(* PLC project actuator, TNI-Software ControlBuild 4.00.17 *)
(* stored: creationDateTime 2005-06-20T11:53:55-01:00 *)

FUNCTION_BLOCK cmd_equipment_library.actuator
  VAR_INPUT  (* CB.group=Modes CB.kind=inputVars *)
    autoMode : BOOL := false;  (* CB.libelle=Automatic mode *)
    manualMode : BOOL := false;  (* CB.libelle=Manual mode *)
  END_VAR
  VAR_INPUT  (* CB.group=Commands CB.kind=inputVars *)
    autoCmd : BOOL := false;  (* CB.libelle=Automatic command of the pump *)
  END_VAR
  VAR_INPUT  (* CB.group=PushButtons CB.kind=inputVars *)
    onPB : BOOL := false;  (* CB.libelle=On pump pushbutton *)
    offPB : BOOL := false;  (* CB.libelle=Off pump pushbutton *)
  END_VAR
  VAR_INPUT  (* CB.kind=inputVars *)
    generalFault : BOOL := false;  (* CB.mnemonicPatternPropertyName=<SY>_DEF_<NU> CB.libelle=General fault of the valve *)
  END_VAR
  VAR_OUTPUT  (* CB.group=Orders CB.kind=outputVars *)
    cmd : BOOL := false;  (* CB.mnemonicPatternPropertyName=cmd<SY><NU> CB.libelle=Command to the pump *)
  END_VAR

(* LD diagram, written out as Structured Text *)
1:
cmd := (autoMode AND autoCmd OR manualMode AND (onPB OR cmd) AND NOT offPB) AND NOT generalFault;
END_FUNCTION_BLOCK
